PROGRAM MAIN
VAR
	fTempSet	: REAL;	
	fbLaudaPro_P20	: FB_LaudaPro_P20;
END_VAR

fbLaudaPro_P20.CommParameters.Ipv4Address := '192.168.0.3';
fbLaudaPro_P20.CommParameters.Port := 54321;
fbLaudaPro_P20.CommParameters.ReadCycle := T#500MS;

fbLaudaPro_P20(fTemperatureSet := fTempSet);

END_PROGRAM

(* stored: Version 1.1.0.1, ProductVersion 3.1.4024.12
   POU MAIN: Id {d83743e1-6877-4583-a383-fad2f5f2df12}, SpecialFunc None *)
